TYPE TMDEStatus :
	(	MDE_Alarm,
		MDE_Production,
		MDE_Standby,
		MDE_Maintenance	);
END_TYPE

(* stored: Version 1.1.0.1, ProductVersion 3.1.4022.12
   DUT TMDEStatus: Id {71e05252-53dd-448f-b4cc-7b23b395f665} *)
